{attribute addProperty BoxType "EL3446-0000-0016"}
{attribute addProperty Id "I1_CurrentAT %I*I1_Current_9D39445A7290I2_CurrentAT %I*I2_Current_9D39445A7290I3_CurrentAT %I*I3_Current_9D39445A7290I4_CurrentAT %I*I4_Current_9D39445A7290I5_CurrentAT %I*I5_Current_9D39445A7290I6_CurrentAT %I*I6_Current_9D39445A7290WcStateAT %I*WcState_F855686C1620InfoDataAT %I*InfoData_0BDED7BF144180"}
{attribute addProperty CRC "1876850235"}
{attribute addProperty SizeInBites "592"}
{attribute addProperty SizeInBytes "74"}
TYPE EL3446_CF284163 :
STRUCT
	{attribute addProperty Name "I1_Current"}
	I1_Current : I1_Current_9D39445A;
	{attribute addProperty Name "I2_Current"}
	I2_Current : I2_Current_9D39445A;
	{attribute addProperty Name "I3_Current"}
	I3_Current : I3_Current_9D39445A;
	{attribute addProperty Name "I4_Current"}
	I4_Current : I4_Current_9D39445A;
	{attribute addProperty Name "I5_Current"}
	I5_Current : I5_Current_9D39445A;
	{attribute addProperty Name "I6_Current"}
	I6_Current : I6_Current_9D39445A;
	{attribute addProperty Name "WcState"}
	WcState : WcState_F855686C;
	{attribute addProperty Name "InfoData"}
	InfoData : InfoData_0BDED7BF;
END_STRUCT
END_TYPE

(* stored: Version 1.2.0.0, ProductVersion 3.1.4024.9
   DUT EL3446_CF284163: Id {1a181e45-1277-4492-9a5d-16d9d2cc4e1e} *)
